{attribute 'qualified_only'}
{attribute 'strict'}
//{attribute 'to_string'}
TYPE EventsEnum :
(
	//standard operation
	//BUNDLE_SENT, // = 0
	BUNDLE_RECEIVED,
	BUNDLE_COMPLETE,
	
	//area complete
	//AREA_1_COMPLETE,
	AREA_2_COMPLETE, //for this area
	//AREA_3_COMPLETE,
	//AREA_4_COMPLETE,
	//AREA_5_COMPLETE,
	//AREA_6_COMPLETE,
	
	//area specific operations
	SECTION_4_COMPLETE,
	SECTION_3_2_1_COMPLETE,
	SECTION_5_COMPLETE,
	SECTION_6_COMPLETE,

	//standard errors
	BACKLOG,
	MACHINE_FAILURE,
	DELAY,
	BUNDLE_EARLY_RECEIVED,
	BUNDLE_LATE_RECEIVED,
	
	//area specific errors
	SECTION_1_FAIL,
	SECTION_2_3_4_FAIL,
	SECTION_5_FAIL,
	SECTION_6_FAIL,
	
	//robots, motors, database, connections, etc
	
	size
);
END_TYPE

(* stored: Version 1.1.0.1, ProductVersion 3.1.4024.11
   EnumerationTextList EventsEnum: Id {7116f09d-954e-4b54-827f-4a9cf285982d} *)
